FUNCTION_BLOCK AX_DEMUX_4 (* AX demultiplexor *)
  (* Standard: 61499-2; Description: Copyright (c) 2024 HR Agrartechnik GmbH This program and the accompanying materials are made available under the terms of the Eclipse Public License 2.0 which is available at https://www.eclipse.org/legal/epl-2.0/ SPDX-License-Identifier: EPL-2.0 *)
  (* Version 1.0, 2024-10-23, Franz Höpfinger, HR Agrartechnik GmbH *)
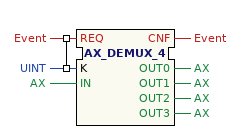
  EVENT_INPUT
    REQ WITH K; (* Set Index K *)
  END_EVENT
  EVENT_OUTPUT
    CNF; (* Confirmation of Set Index K *)
  END_EVENT
  VAR_INPUT
    K : UINT; (* index *)
  END_VAR
  SOCKETS
    IN : AX; (* Input Value to demultiplex *)
  END_SOCKETS
  PLUGS
    OUT0 : AX;
    OUT1 : AX;
    OUT2 : AX;
    OUT3 : AX;
  END_PLUGS
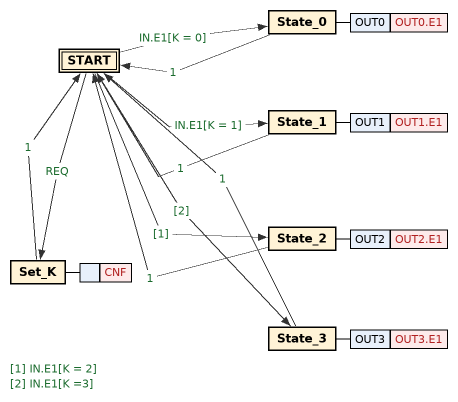
  EC_STATES
    START; (* Initial State *)
    State_0 : OUT0 -> OUT0.E1;
    State_1 : OUT1 -> OUT1.E1;
    Set_K : -> CNF;
    State_2 : OUT2 -> OUT2.E1;
    State_3 : OUT3 -> OUT3.E1;
  END_STATES
  EC_TRANSITIONS
    START TO State_0 := IN.E1[K = 0];
    START TO State_1 := IN.E1[K = 1];
    State_0 TO START := 1;
    State_1 TO START := 1;
    START TO State_2 := IN.E1[K = 2];
    START TO Set_K := REQ;
    Set_K TO START := 1;
    State_2 TO START := 1;
    START TO State_3 := IN.E1[K =3];
    State_3 TO START := 1;
  END_TRANSITIONS
  ALGORITHM OUT0 IN ST:
OUT0.D1 := IN.D1;
  END_ALGORITHM
  ALGORITHM OUT1 IN ST:
OUT1.D1 := IN.D1;
  END_ALGORITHM
  ALGORITHM OUT2 IN ST:
OUT2.D1 := IN.D1;
  END_ALGORITHM
  ALGORITHM OUT3 IN ST:
OUT3.D1 := IN.D1;
  END_ALGORITHM
END_FUNCTION_BLOCK
